{attribute 'qualified_only'}
{attribute 'strict'}
TYPE ESlitDoorPosition :
(
	Unknown := 0,
	Open,
	Close,
	Error
);
END_TYPE

(* stored: Version 1.1.0.1, ProductVersion 3.1.4024.12
   DUT ESlitDoorPosition: Id {8543d742-9f32-4190-b8e6-bb6bcc1dff0a} *)
